Universal Robots PolyScope program: b_zend5.urp

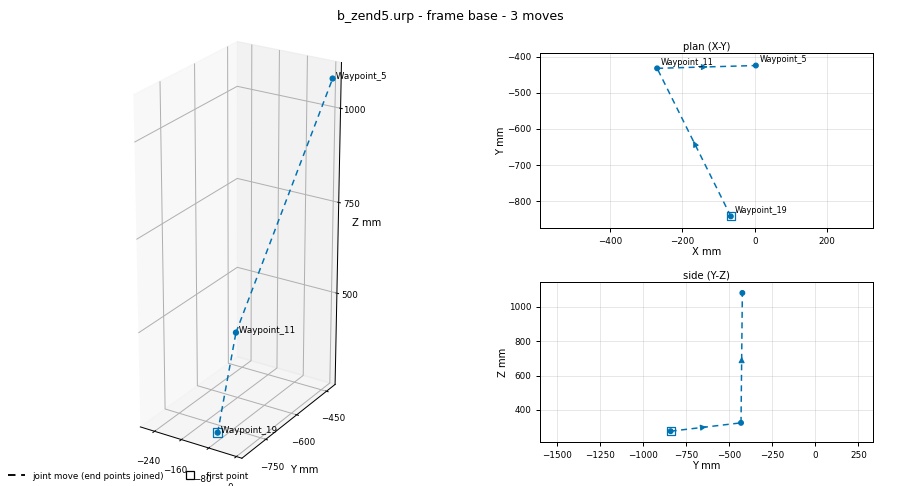
[picture p0: tool path of b_zend5.urp in frame base, 3 of 3 moves have a stored position in this frame; points joined in program order, loops and branches not executed]
Program b_zend5 (installation=default directory=/programs/Burkat_U_Plant createdIn=5.12.6.1102099 lastSavedIn=5.12.6.1102099 robotSerialNumber=20215500597)
Calibrated DH parameters: a=[0.000193, -0.066673, -0.391568, -0.000012, 0.00005, 0]; d=[0.162643, -472.05677, 465.132521, 7.058239, 0.099746, 0.099582]; alpha=[1.571116, 0.00089, 0.003862, 1.569269, -1.569248, 0]; deltaTheta=[0, -1.413394, 7.628392, 0.068187, 0, -0.000001]
Robot Program (runOnlyOnce=true)
  MoveJ speed 60 deg/s, acceleration 80 deg/s^2 (useActiveTCP=true) feature=Base
    Waypoint Waypoint_19: TCP in base x=-66.326 y=-841.615 z=276.687 mm, rx=1.6517 ry=-0.0259 rz=-0.093 rad; joints [71.48, -64.638, 86.648, -17.383, 75.945, -3.629] deg; TCP offset x=0 y=0 z=191.5 mm, rx=0 ry=0 rz=0 rad
    Waypoint Waypoint_11: TCP in base x=-269.994 y=-432.539 z=325.272 mm, rx=1.6722 ry=-0.6368 rz=-0.3794 rad; joints [26.737, -115.333, 124.939, 3.276, 63.256, -0.008] deg
    Waypoint Waypoint_5: TCP in base x=2.907 y=-424.808 z=1080.56 mm, rx=-0.0058 ry=2.215 rz=-2.2169 rad; joints [0.172, -90.171, 0.225, -89.838, 0.52, -0.053] deg
  URCap Gripper (Robotiq_Grippers, Robotiq Inc.) dataModel(position=100.0, force=50.19607843137255, speed=12.274509803921568, positionInDouble=100.0, forceInDouble=50.19607843137255, speedInDouble=12.274509803921568, slaveIds=[9], blocking=true)
